PROGRAM MAIN
VAR
END_VAR

END_PROGRAM

(* stored: Version 1.1.0.1
   POU MAIN: Id {9bacb4b3-46f5-423a-b4d5-1db53caa85af} *)
